// TIA Portal project "TestIS" (V13)

(* hardware
DEVICE "S7300/ET200M station_1"  S7-300 station
   slot 0: "Rail_0"  Rail  6ES7 390-1***0-0AA0
   slot 1: "PS 307 5A_1"  PS 307 5A  6ES7 307-1EA01-0AA0
   slot 2: "PLC-243"  CPU 314C-2 PN/DP  6ES7 314-6EH04-0AB0  V3.3
      slot 2: "PROFINET interface_1"  PN-IO
         slot 1: "Port_1"  Port
         slot 2: "Port_2"  Port
      slot 5: "DI 24/DO 16_1"  DI24/DO16
      slot 6: "AI 5/AO 2_1"  AI5/AO2
      slot 7: "Count_1"  Counter
      slot 8: "Positioning_1"  Positioning
   slot 4: "DI 16x24VDC_1"  DI16 x 24VDC  6ES7 321-1BH02-0AA0
*)

// ===== PLC "PLC-243"  CPU 314C-2 PN/DP =====

VAR_GLOBAL   // PLC tag table "Default tag table"
   "kljuc" AT %I1.2 : Bool;
   "lucka_bos_vidu_kera" AT %Q1.7 : Bool;
   "lucka_levo_rdeca" AT %Q1.4 : Bool;
   "tipka_zgoraj_levo" AT %I1.4 : Bool;
   "tipka_zgoraj_desno" AT %I1.6 : Bool;
   "zelena_tipka" AT %I1.3 : Bool;
   "rumena_leva_lucka" AT %Q1.5 : Bool;
   "vrtljiva_miza_CW" AT %Q0.7 : Bool;
   "vrtljiva_miza_CCW" AT %Q0.6 : Bool;
   "Stevec_za_motorje" AT %C0 : Counter;
   "tipka_spodaj_desno" AT %I1.7 : Bool;
   "tipka_spodaj_levo" AT %I1.5 : Bool;
   "Tag_1" AT %Q1.6 : Bool;
   "izteg" AT %Q1.3 : Bool;
   "krcenje" AT %Q1.2 : Bool;
END_VAR

DATA_BLOCK "gregor"   // DB1
{ S7_Optimized_Access := 'FALSE' }
VERSION : 0.1
   VAR
      poz_1 : Bool;
      poz_2 : Bool;
      SR_lucka : Bool;
      lucka_stanje : Bool;
      stevec_motorji : Word;
      vrtljiva_miza : Bool;
      teleskopska_roka : Bool;
      dvig : Bool;
      prijemalo : Bool;
   END_VAR
BEGIN
END_DATA_BLOCK

DATA_BLOCK "Motorji_izteg_DB"   // DB2
{ S7_Optimized_Access := 'FALSE' }
VERSION : 0.1
// stored: InstanceOfName Motorji_izteg
"Motorji_izteg"
BEGIN
END_DATA_BLOCK

FUNCTION_BLOCK "Motorji_izteg"   // FB1, LAD
{ S7_Optimized_Access := 'FALSE' }
VERSION : 0.1
BEGIN

REGION Network 1
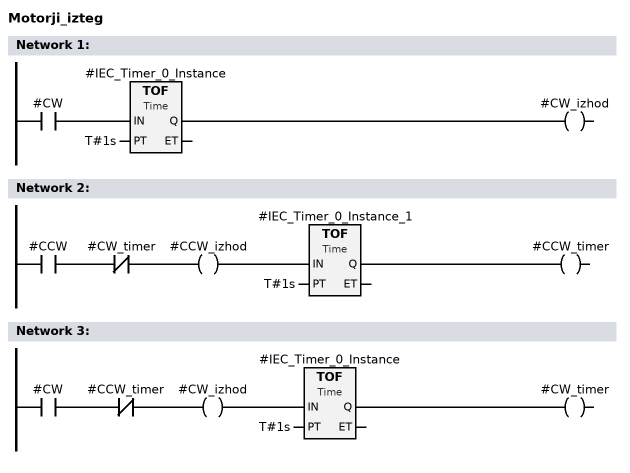
   #IEC_Timer_0_Instance.TOF(IN := #CW, PT := T#1s);
   #CW_izhod := #IEC_Timer_0_Instance.Q;
END_REGION

REGION Network 2
   #CCW_izhod := #CCW AND NOT #CW_timer;
   #IEC_Timer_0_Instance_1.TOF(IN := #CCW_izhod, PT := T#1s);
   #CCW_timer := #IEC_Timer_0_Instance_1.Q;
END_REGION

REGION Network 3
   #CW_izhod := #CW AND NOT #CCW_timer;
   #IEC_Timer_0_Instance.TOF(IN := #CW_izhod, PT := T#1s);
   #CW_timer := #IEC_Timer_0_Instance.Q;
END_REGION
END_FUNCTION_BLOCK

ORGANIZATION_BLOCK "Main"   // OB1, LAD
TITLE = "Main Program Sweep (Cycle)"
{ S7_Optimized_Access := 'FALSE' }
VERSION : 0.1
   VAR_TEMP   // added for the SCL form of the ladder/FBD networks
      _w1 : Bool;
      _w2 : Bool;
   END_VAR
BEGIN

REGION Network 1: Logika_za_lucko
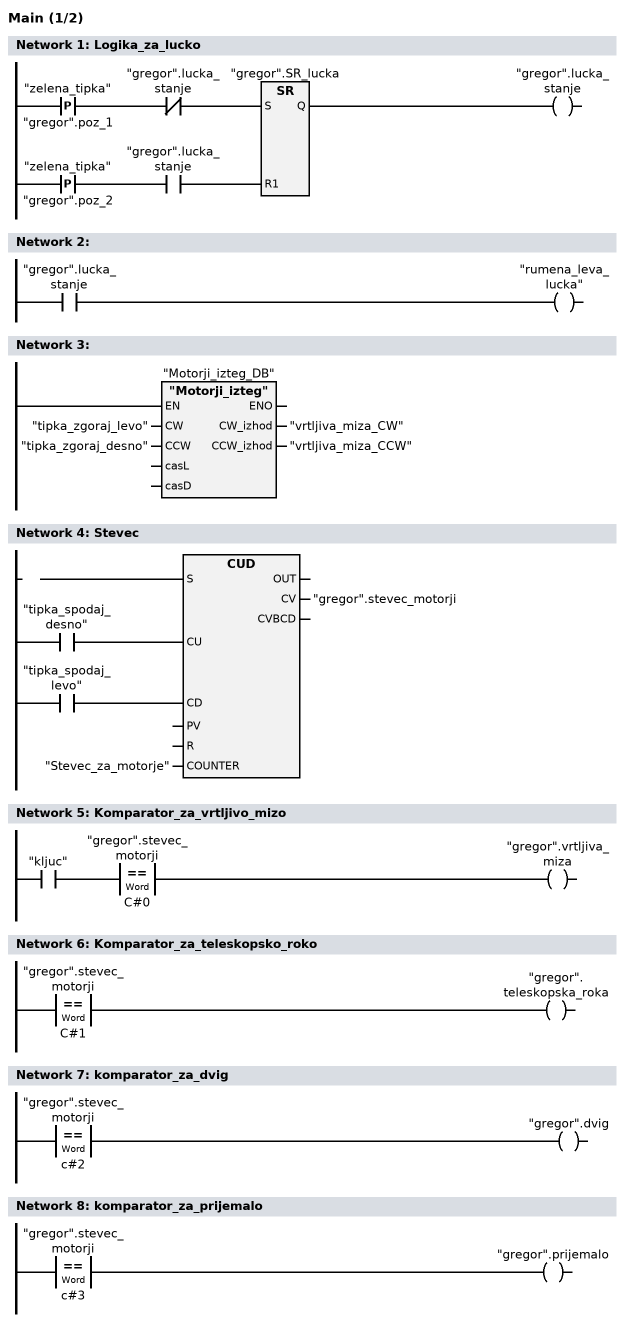
   RUNG wire#powerrail
      P_Contact(operand := "zelena_tipka", bit := "gregor".poz_1)
      I_Contact( "gregor".lucka_stanje )
      S_SR(operand := "gregor".SR_lucka, r1 := wire#w1)
      Coil( "gregor".lucka_stanje )
   END_RUNG
   RUNG wire#powerrail
      P_Contact(operand := "zelena_tipka", bit := "gregor".poz_2)
      Contact( "gregor".lucka_stanje )
   END_RUNG wire#w1
   // the same network as SCL:
   #_w1 := "zelena_tipka" AND NOT "gregor".poz_1;   // rising edge of "zelena_tipka"
   "gregor".poz_1 := "zelena_tipka";
   #_w2 := "zelena_tipka" AND NOT "gregor".poz_2;   // rising edge of "zelena_tipka"
   "gregor".poz_2 := "zelena_tipka";
   IF #_w1 AND NOT "gregor".lucka_stanje THEN
       "gregor".SR_lucka := TRUE;   // SR flip-flop
   END_IF;
   IF #_w2 AND "gregor".lucka_stanje THEN "gregor".SR_lucka := FALSE; END_IF;
   "gregor".lucka_stanje := "gregor".SR_lucka;
END_REGION

REGION Network 2
   RUNG wire#powerrail
      Contact( "gregor".lucka_stanje )
      Coil( "rumena_leva_lucka" )
   END_RUNG
   // the same network as SCL:
   "rumena_leva_lucka" := "gregor".lucka_stanje;
END_REGION

REGION Network 3
   RUNG wire#powerrail
      "Motorji_izteg_DB"(CW := "tipka_zgoraj_levo", CCW := "tipka_zgoraj_desno", casL :=, casD :=, CW_izhod => "vrtljiva_miza_CW", CCW_izhod => "vrtljiva_miza_CCW")
   END_RUNG
   // the same network as SCL:
   "Motorji_izteg_DB"(CW := "tipka_zgoraj_levo",   // "Motorji_izteg"
                      CCW := "tipka_zgoraj_desno",
                      CW_izhod => "vrtljiva_miza_CW",
                      CCW_izhod => "vrtljiva_miza_CCW");
END_REGION

REGION Network 4: Stevec
   // no SCL statement known for Cud: written as a call
   Cud(cu := "tipka_spodaj_desno",
       cd := "tipka_spodaj_levo",
       "counter" := "Stevec_za_motorje",
       cv => "gregor".stevec_motorji);
END_REGION

REGION Network 5: Komparator_za_vrtljivo_mizo
   RUNG wire#powerrail
      Contact( "kljuc" )
      { S7_Templates := "SrcType := Word" } EQ_Contact(in1 := "gregor".stevec_motorji, in2 := C#0)
      Coil( "gregor".vrtljiva_miza )
   END_RUNG
   // the same network as SCL:
   "gregor".vrtljiva_miza := "kljuc" AND ("gregor".stevec_motorji = C#0);
END_REGION

REGION Network 6: Komparator_za_teleskopsko_roko
   RUNG wire#powerrail
      { S7_Templates := "SrcType := Word" } EQ_Contact(in1 := "gregor".stevec_motorji, in2 := C#1)
      Coil( "gregor".teleskopska_roka )
   END_RUNG
   // the same network as SCL:
   "gregor".teleskopska_roka := "gregor".stevec_motorji = C#1;
END_REGION

REGION Network 7: komparator_za_dvig
   RUNG wire#powerrail
      { S7_Templates := "SrcType := Word" } EQ_Contact(in1 := "gregor".stevec_motorji, in2 := c#2)
      Coil( "gregor".dvig )
   END_RUNG
   // the same network as SCL:
   "gregor".dvig := "gregor".stevec_motorji = c#2;
END_REGION

REGION Network 8: komparator_za_prijemalo
   RUNG wire#powerrail
      { S7_Templates := "SrcType := Word" } EQ_Contact(in1 := "gregor".stevec_motorji, in2 := c#3)
      Coil( "gregor".prijemalo )
   END_RUNG
   // the same network as SCL:
   "gregor".prijemalo := "gregor".stevec_motorji = c#3;
END_REGION

REGION Network 10
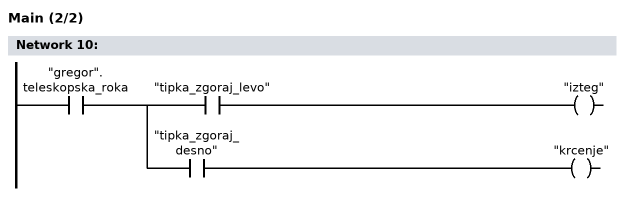
   RUNG wire#powerrail
      Contact( "gregor".teleskopska_roka )
      wire#w1
      Contact( "tipka_zgoraj_levo" )
      Coil( "izteg" )
   END_RUNG
   RUNG wire#w1
      Contact( "tipka_zgoraj_desno" )
      Coil( "krcenje" )
   END_RUNG
   // the same network as SCL:
   "izteg" := "gregor".teleskopska_roka AND "tipka_zgoraj_levo";
   "krcenje" := "gregor".teleskopska_roka AND "tipka_zgoraj_desno";
END_REGION
END_ORGANIZATION_BLOCK